RoboDK station: vector_to_euler_test.rdk

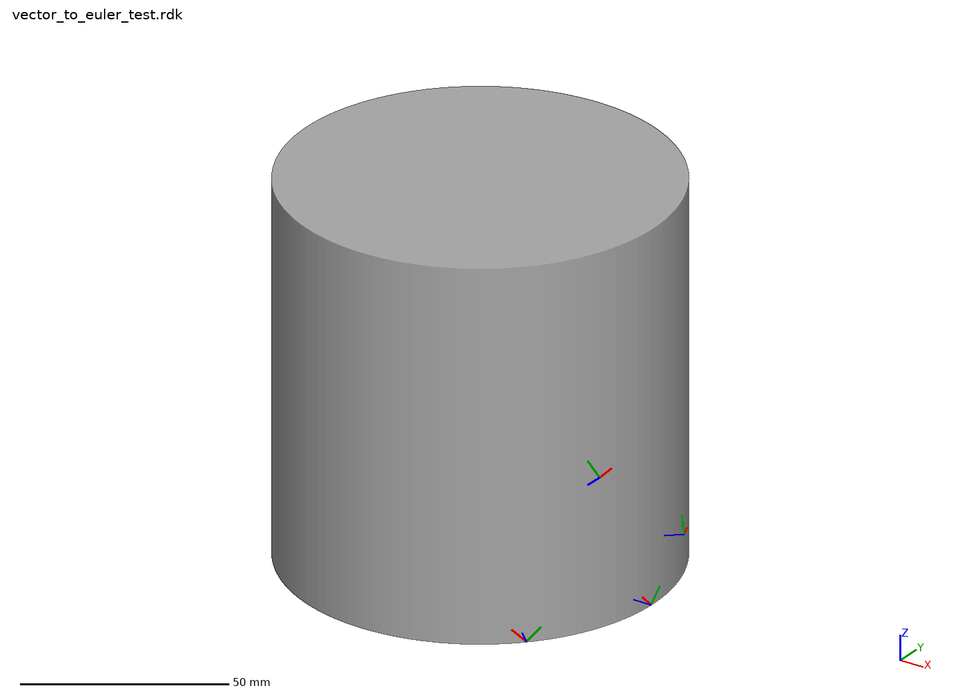
[picture v0: the station drawn from its stored meshes, robots at their saved joint values, targets as dots, program paths as lines]
Station vector_to_euler_test (saved by RoboDK 5.0.0). Poses are relative to the parent item; angles as X-Y-Z fixed-axis rotations.
  - object cylinder50 at (0, 0, 0) mm, size 100 x 100 x 100 mm, geometry from cylinder50.stl
  - frame Frame 1 at (0, 50, 0) mm, rotated rx 90 ry -45 rz 0 deg
  - frame Frame 2 at (34.44, 36.25, 0) mm, rotated rx 90 ry -45 rz -45 deg
  - frame Frame 3 at (50, 0, 0) mm, rotated rx 90 ry -45 rz -90 deg
  - frame Frame 4 at (37, -33.53, 0) mm, rotated rx 90 ry -45 rz -135 deg
  - frame Frame 6 at (0, 1050, 0) mm, rotated rx 0 ry -90 rz -45 deg
    - frame Frame 7 at (0, 0, 0) mm
  - frame Frame 8 at (0, 1070, 0) mm, rotated rx 0 ry -90 rz -45 deg
